RoboDK station: exercise_1.rdk

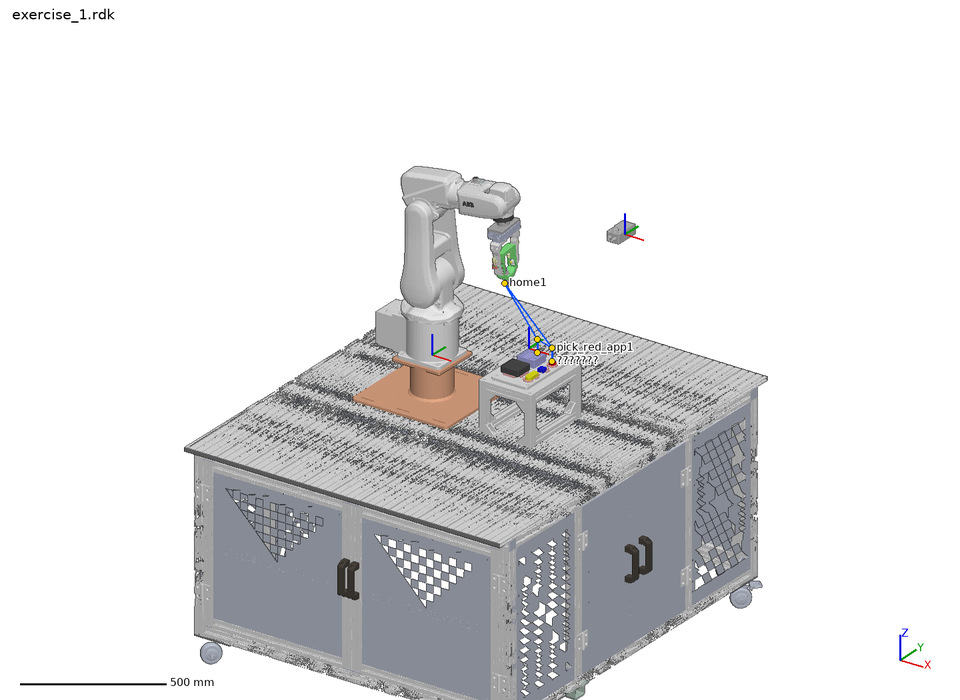
[picture v0: the station drawn from its stored meshes, robots at their saved joint values, targets as dots, program paths as lines]
Station exercise_1 (saved by RoboDK 5.7.1). Poses are relative to the parent item; angles as X-Y-Z fixed-axis rotations.
  - object  at (300, 150, 50) mm, size 220 x 300 x 240 mm, geometry from .stp
  - object  at (382, -48, 89) mm, size 74 x 74 x 28 mm, geometry from .STEP
  - object  at (0, 0, 0) mm, size 1364.5 x 1600 x 1000 mm, geometry from .stp
  - object  at (453, -52, 75) mm, size 24 x 57 x 15 mm, geometry from .stp
  - object  at (453, 10, 75) mm, size 24 x 24 x 15 mm, geometry from .stp
  - frame Frame 2 at (0, 0, 0) mm
    - robot ABB IRB 120-3/0.6: 6 axes, payload 3 kg, reach 580 mm, repeatability 0.01 mm, weight 25 kg
        modified DH rows (alpha deg, a mm, theta deg, d mm): 0, 0, 0, 290; -90, 0, -90, 0; 0, 270, 0, 0; -90, 70, 0, 302; 90, 0, 0, 0; -90, 0, 180, 72
        joint limits [-165, -110, -90, -160, -120, -400] to [165, 110, 70, 160, 120, 400]; home [0, 0, 0, 0, 0, 0]; saved at [2.876, -2.534, -2.625, 2.86, 92.772, -0.394]
      - tool , TCP at (0, 0, 200) mm, size 64.6 x 161.9 x 253.5 mm, geometry from .STEP
    - frame Frame 3 at (0, 1150, 0) mm
      - object SICK-VSPP-5F2113 at (0, 0, 0) mm, size 53 x 116 x 38 mm, geometry from SICK-VSPP-5F2113.stl
    - frame 搬运坐标系 at (300, 150, 50) mm
      - target home1 (Cartesian target) at (2, -150, 308) mm, rotated rx 180 ry 0 rz -180 deg; joints [0, 0, 0, 0, 90, 0] of ABB IRB 120-3/0.6
      - target pick_red_app1 (Cartesian target) at (153, -80, 75) mm, rotated rx 180 ry 0 rz 180 deg; joints [8.784, 38.156, -5.247, 0, 57.091, 8.784] of ABB IRB 120-3/0.6
      - target 红色工件抓取点 (Cartesian target) at (153, -80, 25) mm, rotated rx 180 ry 0 rz 180 deg; joints [8.784, 42.584, -2.314, 0, 49.73, 8.784] of ABB IRB 120-3/0.6
      - target 红色工件预放置点 (Cartesian target) at (97, -87, 95) mm, rotated rx 180 ry 0 rz 180 deg; joints [9.017, 25.21, 10.07, 0, 54.72, 9.017] of ABB IRB 120-3/0.6
      - target 红色工件放置点 (Cartesian target) at (97, -87, 45) mm, rotated rx 180 ry 0 rz 180 deg; joints [9.017, 29.919, 13.562, 0, 46.519, 9.017] of ABB IRB 120-3/0.6
  - program 示例1 (14 instructions, listed below)
  - Python program python_test_1 (listed below)
  - Python program Prog3 (listed below)
  - Python program test_2 (listed below)
  - Python program RL_SAC (listed below)
  - object  at (453, 70, 75) mm, size 24 x 24 x 15 mm, geometry from .stp
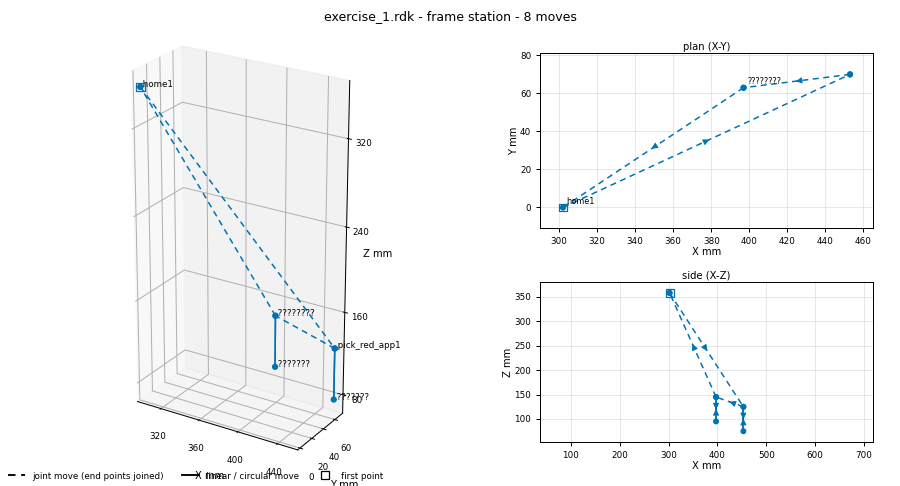
[picture p0: tool path of exercise_1.rdk in frame station, 8 of 8 moves have a stored position in this frame; points joined in program order, loops and branches not executed]

--- program 示例1 (robot ABB IRB 120-3/0.6) ---
  设置参考号: 搬运坐标系
  设置工具: 吸盘工具 at (0, 0, 200) mm
  设置速度（10.0 mm/s)
  替换物体
  MoveJ (首页) -> target home1
  MoveJ (红色工件预抓取点) -> target pick_red_app1
  MoveL (红色工件抓取点)
  附加到吸盘工具
  MoveL (红色工件预抓取点) -> target pick_red_app1
  MoveJ (红色工件预放置点)
  MoveL (红色工件放置点)
  分离于吸盘工具
  MoveL (红色工件预放置点)
  MoveJ (首页) -> target home1

--- Python program python_test_1 ---
from robolink import *    # RoboDK API
from robodk import *      # Robot toolbox
RDK = Robolink()
pose = eye()
##########定义对象##########
robot = RDK.Item('ABB IRB 120-3/0.6')
tool = RDK.Item('吸盘工具')
referencing_frame = RDK.Item('搬运坐标系')
red_part = RDK.Item('红色工件')
blue_part = RDK.Item('蓝色工件')
yellow_part = RDK.Item('黄色工件')
cover = RDK.Item('端盖')

##########定义目标点##########

pick_red = transl(153,-80,25)*rotz(pi)*rotx(pi)
put_red_app = transl(97,-87,25)*rotz(pi)*rotx(pi)
put_red = transl(97,-87,45)*rotz(pi)*rotx(pi)

##########定义初始化函数#########
def init():
    red_part.setPose(transl(453,70,75))
    yellow_part.setPose(transl(453,-52,75))
    blue_part.setPose(transl(453,10,75))
    cover.setPose(transl(382,-48,89))

##########仿真程序##########
init()
robot.setPoseTool(tool)
robot.setPoseFrame(referencing_frame)
robot.setSpeed(20,20,-1,-1)
print(robot.Joints())

robot.MoveJ(home_1)
robot.MoveJ(pick_red_app_1)
robot.MoveL(pick_red)
tool.AttachClosest()
pause(0.2)
robot.MoveL(pick_red_app_1)
robot.MoveJ(put_red_app)
robot.MoveL(put_red)
tool.DetachAll()
pause(0.2)
robot.MoveL(put_red_app)
robot.MoveJ(home_1)

--- Python program Prog3 ---
import gym
import numpy as np
from stable_baselines3 import SAC,DQN
from stable_baselines3.common.vec_env import DummyVecEnv
from robolink import *    # RoboDK API
from robodk import *      # Robot toolbox
import  torch

num_epochs = 100  # 训练回合数
capacity = 500  # 经验池容量
min_size = 200  # 经验池训练容量
batch_size = 64
n_hiddens = 64
actor_lr = 1e-3  # 策略网络学习率
critic_lr = 1e-2  # 价值网络学习率
alpha_lr = 1e-2  # 课训练变量的学习率
target_entropy = -1
tau = 0.005  # 软更新参数
gamma = 0.9  # 折扣因子
device = torch.device('cuda') if torch.cuda.is_available() else torch.device('cpu')

# 初始化RoboDK环境
class RoboDKEnv(gym.Env):
    def __init__(self):
        self.RDK = Robolink()
        self.robot = self.RDK.Item('ABB IRB 120-3/0.6')
        self.tool = self.RDK.Item('吸盘工具')
        self.referencing_frame = self.RDK.Item('搬运坐标系')
        self.red_part = self.RDK.Item('红色工件')
        self.blue_part = self.RDK.Item('蓝色工件')
        self.yellow_part = self.RDK.Item('黄色工件')
        self.cover = self.RDK.Item('端盖')
        self.home_1 = self.RDK.Item('home1')
        self.home_2 = self.RDK.Item('home2')
        self.home_3 = self.RDK.Item('home3')
        self.home_4 = self.RDK.Item('home4')
        self.pick_red_app_1 = self.RDK.Item('pick_red_app1')
        self.pick_red_app_2 = self.RDK.Item('pick_red_app2')
        self.pick_red_app_3 = self.RDK.Item('pick_red_app3')
        self.pick_red_app_4 = self.RDK.Item('pick_red_app4')
        self.pick_red = transl(153,-80,25)*rotz(pi)*rotx(pi)
        self.put_red_app = transl(97,-87,25)*rotz(pi)*rotx(pi)
        self.put_red = transl(97,-87,45)*rotz(pi)*rotx(pi)
        self.action_space = gym.spaces.Box(low=np.array([453, -52, 10, 97, -87, 25]),
                                            high=np.array([453, 70, 75, 153, -80, 25]))   # home和pick_red_app positions
        self.observation_space = gym.spaces.Box(low=-np.inf, high=np.inf, shape=(1,)) # 修改为适当的观察空间
        self.reward_range = (-np.inf, np.inf)
        self.done = False
        self.current_step = 0

    def reset(self):
        self.done = False
        self.current_step = 0
        self.init()
        return np.array([0])

    def step(self, action):
        home_action = action[:3]
        pick_red_app_action = action[3:]
        self.move_robot(home_action, pick_red_app_action)
        self.current_step += 1
        if self.current_step == 8:  # 假设一个回合有8个动作（4个home选择 + 4个pick_red_app选择）
            self.done = True
        reward = self.calculate_reward()
        return np.array([0]), reward, self.done, {}

    def move_robot(self, home_action, pick_red_app_action):
        # 移动机器人
        home_pos = [self.home_1, self.home_2, self.home_3, self.home_4][np.argmax(home_action)]
        pick_red_app_pos = [self.pick_red_app_1, self.pick_red_app_2, self.pick_red_app_3, self.pick_red_app_4][np.argmax(pick_red_app_action)]
        self.robot.MoveJ(home_pos)
        self.robot.MoveJ(pick_red_app_pos)

    def calculate_reward(self):
        # 计算奖励
        # 这里简单地假设回合完成时间越短，奖励越高
        return -self.current_step

    def init(self):
        # 初始化机器人位置
        pass  # 这里可以根据需要初始化机器人的位置

# 创建环境
env = RoboDKEnv()
env = DummyVecEnv([lambda: env])

# 使用SAC算法训练智能体
# model = SAC("MlpPolicy", env, verbose=1)
model = DQN("MlpPolicy",env, verbose=1,gamma=gamma,tau=tau,device="cuda",tensorboard_log="log/")

model.learn(total_timesteps=10000)

# 保存训练好的模型
model.save("sac_robot_model")

--- Python program test_2 ---
from robolink import *  # RoboDK API
from robodk import *  # Robot toolbox
import numpy as np

RDK = Robolink()
pose = eye()
##########定义对象##########
robot = RDK.Item('ABB IRB 120-3/0.6')
tool = RDK.Item('吸盘工具')
referencing_frame = RDK.Item('搬运坐标系')
red_part = RDK.Item('红色工件')
blue_part = RDK.Item('蓝色工件')
yellow_part = RDK.Item('黄色工件')
cover = RDK.Item('端盖')

##########定义目标点##########
home_1 = RDK.Item('home1')
home_2 = RDK.Item('home2')
home_3 = RDK.Item('home3')
home_4 = RDK.Item('home4')
home_5 = RDK.Item('home5')
home_6 = RDK.Item('Target 13')  # 新的目标点
pick_red_app_1 = RDK.Item('pick_red_app1')
pick_red_app_2 = RDK.Item('pick_red_app2')
pick_red_app_3 = RDK.Item('pick_red_app3')
pick_red_app_4 = RDK.Item('pick_red_app4')

pick_red = transl(153, -80, 25) * rotz(pi) * rotx(pi)
put_red_app = transl(97, -87, 25) * rotz(pi) * rotx(pi)
put_red = transl(97, -87, 45) * rotz(pi) * rotx(pi)


##########定义初始化函数#########
def init():
    red_part.setPose(transl(453, 70, 75))
    yellow_part.setPose(transl(453, -52, 75))
    blue_part.setPose(transl(453, 10, 75))
    cover.setPose(transl(382, -48, 89))


##########仿真程序##########
init()
robot.setPoseTool(tool)
robot.setPoseFrame(referencing_frame)
robot.setSpeed(20, 20, -1, -1)
print(robot.Joints())

import time

import numpy as np


def pose_to_rot_mat(pose):
    # Convert pose to rotation matrix
    rot_mat = np.array([[pose[0, 0], pose[0, 1], pose[0, 2]],
                        [pose[1, 0], pose[1, 1], pose[1, 2]],
                        [pose[2, 0], pose[2, 1], pose[2, 2]]])
    return rot_mat


def pieper_inverse_kinematics(pose):
    # Extract position and rotation from pose
    position = pose.Pos()
    rotation = pose_to_rot_mat(pose)

    # Initialize joint angles
    joint_angles = [0] * 6

    # Calculate joint angles
    # Joint 1 (theta1)
    joint_angles[0] = np.arctan2(position[1], position[0])

    # Joint 3 (theta3)
    D = (position[0] ** 2 + position[1] ** 2 + (position[2] - 72) ** 2 - 70 ** 2 - 302 ** 2 - 270 ** 2) / (2 * 70 * 302)
    if -1 <= D <= 1:
        joint_angles[2] = np.arctan2(-np.sqrt(1 - D ** 2), D)
    else:
        # Handle cases where D is out of valid range
        joint_angles[2] = 0  # Set joint angle to default value

    # Joint 2 (theta2)
    alpha = np.arctan2(position[2] - 72, np.sqrt(position[0] ** 2 + position[1] ** 2))
    beta = np.arctan2(302 * np.sin(joint_angles[2]), 70 + 302 * np.cos(joint_angles[2]))
    joint_angles[1] = np.pi / 2 - alpha - beta

    # Joint 4, 5, 6 (theta4, theta5, theta6)
    R03 = np.array([[np.cos(joint_angles[0]) * np.cos(joint_angles[1] + joint_angles[2]), -np.sin(joint_angles[0]),
                     np.cos(joint_angles[0]) * np.sin(joint_angles[1] + joint_angles[2])],
                    [np.sin(joint_angles[0]) * np.cos(joint_angles[1] + joint_angles[2]), np.cos(joint_angles[0]),
                     np.sin(joint_angles[0]) * np.sin(joint_angles[1] + joint_angles[2])],
                    [-np.sin(joint_angles[1] + joint_angles[2]), 0, np.cos(joint_angles[1] + joint_angles[2])]])

    R36 = np.dot(np.linalg.inv(R03), rotation)
    joint_angles[3] = np.arctan2(R36[2, 1], R36[2, 2])
    joint_angles[3] = -25.1
    joint_angles[4] = -np.arctan2(-R36[2, 0], np.sqrt(R36[0, 0] ** 2 + R36[1, 0] ** 2))
    joint_angles[5] = np.arctan2(R36[1, 0], R36[0, 0])

    return joint_angles


robot_item_list = [robot]
joints_list = []
count = 0
# 从0度到90度，每秒变化10度
for angle in range(0, 91, 10):
    count += 1
    current_joint_angles = [angle, -0.000, 0.000, 0.000, 90.000, -0.000]
    joints_list.append(current_joint_angles)

    RDK.setJoints(robot_item_list, [current_joint_angles])

    # robodk自带的旋转矩阵计算
    if angle % 30 == 0:
        print("Current joint angles:\n", robot.Joints())
        print("Current Rotation Matrix:\n", Mat(robot.SolveFK(current_joint_angles)))

        # DH表得出数据进行选择矩阵计算
        # DH参数
        theta = current_joint_angles
        d = [290, 0, 0, 302, 0, 72]
        a = [0, 270, 70, 0, 0, 0]
        alpha = [np.radians(-90), np.radians(0), np.radians(-90), np.radians(0), np.radians(-90), np.radians(0)]


        # 定义选择矩阵函数
        def compute_transform_matrix(theta, d, a, alpha):
            return np.array([
                [np.cos(theta), -np.sin(theta) * np.cos(alpha), np.sin(theta) * np.sin(alpha), a * np.cos(theta)],
                [np.sin(theta), np.cos(theta) * np.cos(alpha), -np.cos(theta) * np.sin(alpha), a * np.sin(theta)],
                [0, np.sin(alpha), np.cos(alpha), d],
                [0, 0, 0, 1]
            ])


        # 计算各个选择矩阵
        A_0_1 = compute_transform_matrix(theta[0], d[0], a[0], alpha[0])
        A_1_2 = compute_transform_matrix(theta[1], d[1], a[1], alpha[1])
        A_2_3 = compute_transform_matrix(theta[2], d[2], a[2], alpha[2])
        A_3_4 = compute_transform_matrix(theta[3], d[3], a[3], alpha[3])
        A_4_5 = compute_transform_matrix(theta[4], d[4], a[4], alpha[4])
        A_5_6 = compute_transform_matrix(theta[5], d[5], a[5], alpha[5])

        # 计算最终选择矩阵
        A_0_6 = np.dot(A_0_1, np.dot(A_1_2, np.dot(A_2_3, np.dot(A_3_4, np.dot(A_4_5, A_5_6)))))

# 使用逆运动学求解home_6的关节角度位置
home_6_pose = home_6.Pose()
home_6_xyzwpr = Pose_2_TxyzRxyz(home_6_pose)
target_joint_angles_DK = robot.SolveIK(home_6_pose)
target_joint_angles = pieper_inverse_kinematics(home_6.Pose())
for i in range(len(target_joint_angles)):
    if i < 3:
        target_joint_angles[i] *= 50  # 将每个关节角度乘以
    #    else:
    #       target_joint_angles[i] *= i*20
    elif i == 4:
        target_joint_angles[i] *= i * i * 20
    elif i == 5:
        target_joint_angles[i] *= i * i * 5

print("Home 6 Pose (XYZWPR):\n", home_6_xyzwpr)

print("Pieper Home 6 Joint Angles:\n", target_joint_angles)

print("RoboDK Home 6 Joint Angles:\n", target_joint_angles_DK)

RDK.setJoints(robot_item_list, [target_joint_angles_DK])
print("**RoboDK Joint Angles:\n", robot.Joints())

time.sleep(2)
RDK.setJoints(robot_item_list, [target_joint_angles])
print("**Pieper Joint Angles:\n", robot.Joints())

--- Python program RL_SAC ---
import gym
from gym import spaces
import numpy as np
from robolink import *    # RoboDK API
from robodk import *      # Robot toolbox
import torch
from stable_baselines3 import SAC

# 连接到RoboDK
RDK = Robolink()

# 定义机械臂和其他对象
robot = RDK.Item('ABB IRB 120-3/0.6')
tool = RDK.Item('吸盘工具')
referencing_frame = RDK.Item('搬运坐标系')
red_part = RDK.Item('红色工件')
blue_part = RDK.Item('蓝色工件')
yellow_part = RDK.Item('黄色工件')
cover = RDK.Item('端盖')

# 定义目标点
home_1 = RDK.Item('home1')
pick_red_app_1 = RDK.Item('pick_red_app1')
put_red_app = transl(97, -87, 25) * rotz(pi) * rotx(pi)
put_red = transl(97, -87, 45) * rotz(pi) * rotx(pi)

# 定义抓取和放置点的关节角度
PICK_JOINTS = np.array([8.784176, 42.583797, -2.314112, 0.000000, 49.730315, 8.784176])
PUT_JOINTS = np.array([9.017088, 29.918624, 13.562401, 0.000000, 46.518975, 9.017088])

# 折扣因子
GAMMA = 1

# 初始化机械臂位置
def init():
    red_part.setPose(transl(453, 70, 75))
    yellow_part.setPose(transl(453, -52, 75))
    blue_part.setPose(transl(453, 10, 75))
    cover.setPose(transl(382, -48, 89))
    robot.setPoseTool(tool)
    robot.setPoseFrame(referencing_frame)
    robot.setSpeed(20, 20, -1, -1)

class PickPlaceEnv(gym.Env):
    def __init__(self):
        super(PickPlaceEnv, self).__init__()
        self.action_space = spaces.Box(low=-1, high=1, shape=(6,), dtype=np.float32)
        self.observation_space = spaces.Box(low=-np.inf, high=np.inf, shape=(12,), dtype=np.float32)
        init()
        self.step_count = 0
        self.subtask = 1  # 初始位置到抓取位置为子任务1，抓取到放置位置为子任务2

    def reset(self):
        init()
        self.robot = robot
        self.robot.MoveJ(home_1)
        self.step_count = 0
        self.subtask = 1
        return self._get_obs()

    def _get_obs(self):
        joints = self.robot.Joints().tolist()
        red_position = list(red_part.Pose().Pos())
        observation = joints + red_position + [0] * (12 - len(joints) - len(red_position))
        return np.array(observation, dtype=np.float32)

    def step(self, action):
        action = np.clip(action, self.action_space.low, self.action_space.high)
        current_joints = np.array(self.robot.Joints().tolist())
        new_joints = (current_joints + action).tolist()

        try:
            self.robot.MoveJ(new_joints)
        except TargetReachError:
            reward = -100
            done = True
            return self._get_obs(), reward, done, {}

        end_effector_pos = list(self.robot.PoseTool().Pos())
        red_pos = list(red_part.Pose().Pos())
        reward = -np.linalg.norm(np.array(end_effector_pos) - np.array(red_pos))

        if self.subtask == 1:
            if self._is_near_joints(PICK_JOINTS):
                self.robot.MoveL(pick_red_app_1)
                self.tool.AttachClosest()
                pause(2)
                reward = 100
                self.subtask = 2
        elif self.subtask == 2:
            reward = -np.linalg.norm(np.array(end_effector_pos) - np.array(put_red.Pos()))
            if self._is_near_joints(PUT_JOINTS):
                self.robot.MoveL(put_red_app)
                self.tool.DetachAll()
                pause(2)
                self.robot.MoveJ(home_1)
                reward = 200
                done = True
                return self._get_obs(), reward, done, {}

        self.step_count += 1
        reward *= GAMMA ** self.step_count
        done = False
        return self._get_obs(), reward, done, {}

    def _is_near_joints(self, target_joints, threshold=5.0):
        current_joints = np.array(self.robot.Joints().tolist())
        return np.linalg.norm(current_joints - target_joints) < threshold

    def render(self, mode='human'):
        pass

env = PickPlaceEnv()

# 使用SAC算法进行训练
print('device is : {}'.format(torch.cuda.is_available()))
device = torch.device("cuda" if torch.cuda.is_available() else "cpu")
model = SAC('MlpPolicy', env, verbose=1, device=device)
model.learn(total_timesteps=20000)
model.save("D:/work/learning/roboDK_learning/sac_robodk_red_pick")

# 测试训练好的模型
model = SAC.load("D:/work/learning/roboDK_learning/sac_robodk_red_pick")
obs = env.reset()
for _ in range(1000):
    action, _states = model.predict(obs)
    obs, rewards, dones, info = env.step(action)
    if dones:
        obs = env.reset()
